PROGRAM MAIN
VAR
	power1,power2,power3,power4: MC_Power;
	axis1,axis2,axis3,axis4: AXIS_REF;
	power1_output,power2_output,power3_output,power4_output:ST_McOutputs;
	

	
	
	move_abs: MC_MoveAbsolute;
	init_pos: LREAL;
	move_init_output:ST_McOutputs;
	
	SetPointGenEnable,SetPointGenEnable1,SetPointGenEnable2,SetPointGenEnable3: MC_ExtSetPointGenEnable;
	SetPointGenDisable,SetPointGenDisable1,SetPointGenDisable2,SetPointGenDisable3: MC_ExtSetPointGenDisable;
	SetPointGenEnable_output,SetPointGenDisable_output,SetPointGenEnable_output1,SetPointGenDisable_output1,SetPointGenEnable_output2,SetPointGenDisable_output2,SetPointGenEnable_output3,SetPointGenDisable_output3:ST_McOutputs;	
	enable,disable:BOOL;
	
	reset_output:ST_McOutputs;
	axis_Reset: MC_Reset;
	
	gen_state:state;
	
	position: LREAL;
	velocity: LREAL;
	direction: DINT;	
	acceleration: LREAL;
	t:LREAL:=0;

	n:UINT:=0;
	a:LINT;
	
	pos1,pos2,pos3,pos4:LREAL;
	acc1,acc2,acc3,acc4:LREAL;
	velo1,velo2,velo3,velo4:LREAL;
	dir: DINT:=1;
	inpos:BOOL:=1;
	flag:UINT:=0;

	flag1: INT;
	ADS_Array: ARRAY[0..12] OF UINT;
	ADS_ParaArray: ARRAY[0..11] OF UINT;
	avar:LREAL;
END_VAR

axis1();(*更新轴状态*)
axis2();(*更新轴状态*)
axis3();(*更新轴状态*)
axis4();(*更新轴状态*)
axis1.ReadStatus();
axis2.ReadStatus();
axis3.ReadStatus();
axis4.ReadStatus();
power();
setpositionGen();
reset();

//move_init();
//TCP/IP receive data
IF NOT GVL.rec_busy THEN
	GVL.bReceive:=TRUE;
END_IF
TCPServer();
IF GVL.number_recdata<>0 THEN
	gen_state:=gen_enable;
	GVL.number_recdata:=0;
	IF GVL.Data_receive[1]>16#7F THEN 
	   GVL.Data_receive[1]:=GVL.Data_receive[1] AND 16#7F;
 	   flag:=1;	
	END_IF
	pos1:=GVL.Data_receive[1];
	pos1:=pos1*256;
	pos1:=(pos1+GVL.Data_receive[2])/10;
	IF flag=1 THEN
		pos1:=-pos1;
		flag:=0;
	END_IF
	velo1:=GVL.Data_receive[3];
	velo1:=velo1*256;
	velo1:=(velo1+GVL.Data_receive[4])/10;
	acc1:=GVL.Data_receive[5];
	acc1:=acc1*256;
	acc1:=(acc1+GVL.Data_receive[6])/10;
	
	IF GVL.Data_receive[7]>16#7F THEN 
	   GVL.Data_receive[7]:=GVL.Data_receive[7] AND 16#7F;
 	   flag:=1;	
	END_IF
	pos2:=GVL.Data_receive[7];
	pos2:=pos2*256;
	pos2:=(pos2+GVL.Data_receive[8])/10;
	IF flag=1 THEN
		pos2:=-pos2;
		flag:=0;
	END_IF
	velo2:=GVL.Data_receive[9];
	velo2:=velo2*256;
	velo2:=(velo2+GVL.Data_receive[10])/10;
	acc2:=GVL.Data_receive[11];
	acc2:=acc2*256;
	acc2:=(acc2+GVL.Data_receive[12])/10;
	
	IF GVL.Data_receive[13]>16#7F THEN 
	   GVL.Data_receive[13]:=GVL.Data_receive[13] AND 16#7F;
 	   flag:=1;	
	END_IF
	pos3:=GVL.Data_receive[13];
	pos3:=pos3*256;
	pos3:=(pos3+GVL.Data_receive[14])/10;
	IF flag=1 THEN
		pos3:=-pos3;
		flag:=0;
	END_IF
	velo3:=GVL.Data_receive[15];
	velo3:=velo3*256;
	velo3:=(velo3+GVL.Data_receive[16])/10;
	acc3:=GVL.Data_receive[17];
	acc3:=acc3*256;
	acc3:=(acc3+GVL.Data_receive[18])/10;
	
	IF GVL.Data_receive[19]>16#7F THEN 
	   GVL.Data_receive[19]:=GVL.Data_receive[19] AND 16#7F;
 	   flag:=1;	
	END_IF
	pos4:=GVL.Data_receive[19];
	pos4:=pos4*256;
	pos4:=(pos4+GVL.Data_receive[20])/10;
	IF flag=1 THEN
		pos4:=-pos4;
		flag:=0;
	END_IF
	velo4:=GVL.Data_receive[21];
	velo4:=velo4*256;
	velo4:=(velo4+GVL.Data_receive[22])/10;
	acc4:=GVL.Data_receive[23];
	acc4:=acc4*256;
	acc4:=(acc4+GVL.Data_receive[24])/10;
END_IF

//ADS receive data
IF ADS_Array[12]=1 THEN
	ADS_Array[12]:=0;
	gen_state:=gen_enable;
	pos1:=ADS_Array[0];
	pos1:=pos1/10;
	velo1:=ADS_Array[1];
	velo1:=velo1/10;
	acc1:=ADS_Array[2];
	acc1:=acc1/10;
	pos2:=ADS_Array[3];
	pos2:=pos2/10;
	velo2:=ADS_Array[4];
	velo2:=velo2/10;
	acc2:=ADS_Array[5];
	acc2:=acc2/10;
	pos3:=ADS_Array[6];
	pos3:=pos3/10;
	velo3:=ADS_Array[7];
	velo3:=velo3/10;
	acc3:=ADS_Array[8];
	acc3:=acc3/10;
	pos4:=ADS_Array[9];
	pos4:=pos4/10;
	velo4:=ADS_Array[10];
	velo4:=velo4/10;
	acc4:=ADS_Array[11];
	acc4:=acc4/10;
END_IF
//ADS updata
avar:=axis1.NcToPlc.ActPos;  //位置
avar:=avar*10;
ADS_ParaArray[0]:= TO_UINT(avar);
avar:=axis1.NcToPlc.Actvelo;  //速度
avar:=avar*10;
ADS_ParaArray[1]:=TO_UINT(avar);
avar:=axis1.NcToPlc.ActAcc;  //加速度
avar:=avar*10;
ADS_ParaArray[2]:=TO_UINT(avar);

avar:=axis2.NcToPlc.ActPos;  //位置
avar:=avar*10;
ADS_ParaArray[3]:= TO_UINT(avar);
avar:=axis2.NcToPlc.Actvelo;  //速度
avar:=avar*10;
ADS_ParaArray[4]:=TO_UINT(avar);
avar:=axis2.NcToPlc.ActAcc;  //加速度
avar:=avar*10;
ADS_ParaArray[5]:=TO_UINT(avar);

avar:=axis3.NcToPlc.ActPos;  //位置
avar:=avar*10;
ADS_ParaArray[6]:= TO_UINT(avar);
avar:=axis3.NcToPlc.Actvelo;  //速度
avar:=avar*10;
ADS_ParaArray[7]:=TO_UINT(avar);
avar:=axis3.NcToPlc.ActAcc;  //加速度
avar:=avar*10;
ADS_ParaArray[8]:=TO_UINT(avar);

avar:=axis4.NcToPlc.ActPos;  //位置
avar:=avar*10;
ADS_ParaArray[9]:= TO_UINT(avar);
avar:=axis4.NcToPlc.Actvelo;  //速度
avar:=avar*10;
ADS_ParaArray[10]:=TO_UINT(avar);
avar:=axis4.NcToPlc.ActAcc;  //加速度
avar:=avar*10;
ADS_ParaArray[11]:=TO_UINT(avar);

CASE gen_state OF
	init:
		power1.Enable:=FALSE;
		power2.Enable:=FALSE;
		power3.Enable:=FALSE;
		power4.Enable:=FALSE;
		SetPointGenEnable.Execute:=FALSE;
		SetPointGenDisable.Execute:=FALSE;
		SetPointGenEnable1.Execute:=FALSE;
		SetPointGenDisable1.Execute:=FALSE;
		SetPointGenEnable2.Execute:=FALSE;
		SetPointGenDisable2.Execute:=FALSE;
		SetPointGenEnable3.Execute:=FALSE;
		SetPointGenDisable3.Execute:=FALSE;
		axis_Reset.Execute:=FALSE;
		gen_state:=gen_power;
			
	gen_power:
		power1.Enable:=TRUE;
		power2.Enable:=TRUE;
		power3.Enable:=TRUE;
		power4.Enable:=TRUE;
		IF power1_output.Done AND power2_output.Done AND power3_output.Done AND power4_output.Done THEN
			gen_state:=gen_move;
		END_IF
		IF axis1.Status.Error OR axis2.Status.Error OR axis3.Status.Error OR axis4.Status.Error THEN
			gen_state := gen_error;
		END_IF
		
	gen_move:
		//	gen_state:=gen_enable;
	gen_enable:

		setpointgenenable.Execute:=TRUE;
		setpointgenenable1.Execute:=TRUE;
		setpointgenenable2.Execute:=TRUE;
		setpointgenenable3.Execute:=TRUE;
		IF SetPointGenEnable.Enabled AND SetPointGenEnable1.Enabled AND SetPointGenEnable2.Enabled AND SetPointGenEnable3.Enabled AND inpos THEN
			flag:=1;
		END_IF

		IF flag=1 THEN
			gen_state:=gen_move;
			IF velo1>1 THEN
				MC_ExtSetPointGenFeed(
					Position:= pos1,		
					Velocity:= velo1, 
					Acceleration:=acc1, 
					Direction:= dir,
					Axis:= axis1);	
			END_IF
			IF velo2>1 THEN
				MC_ExtSetPointGenFeed(
					Position:= pos2,		
					Velocity:= velo2, 
					Acceleration:=acc2, 
					Direction:= dir,
					Axis:= axis2);	
			END_IF
			IF velo3>1 THEN
				MC_ExtSetPointGenFeed(
					Position:= pos3,		
					Velocity:= velo3, 
					Acceleration:=acc3, 
					Direction:= dir,
					Axis:= axis3);
			END_IF	
			IF velo4>1 THEN
				MC_ExtSetPointGenFeed(
					Position:= pos4,		
					Velocity:= velo4, 
					Acceleration:=acc4, 
					Direction:= dir,
					Axis:= axis4);
			END_IF	
		END_IF
		
	//	IF axis1.Status.InTargetPosition AND axis2.Status.InTargetPosition AND axis3.Status.InTargetPosition AND axis4.Status.InTargetPosition AND flag=0 THEN
	//		inpos:=TRUE;
	//	END_IF
		
		IF flag=1 THEN
			flag:=0;
		END_IF

		IF axis1.Status.Error THEN
			gen_state := gen_error;
		END_IF
	
	gen_error:
		SetPointGenEnable.Execute:=FALSE;
		SetPointGenDisable.Execute := SetPointGenEnable.Enabled;	
		SetPointGenEnable1.Execute:=FALSE;
		SetPointGenDisable1.Execute := SetPointGenEnable1.Enabled;
		IF NOT axis1.Status.Coupled THEN
			IF axis1.Status.Error THEN
				gen_state := gen_reset;	
			ELSE
				gen_state := init;
			END_IF
		END_IF
	
	gen_reset:
		axis_Reset.Execute := TRUE;
		SetPointGenDisable.Execute:=FALSE;
		SetPointGenDisable1.Execute:=FALSE;
			
			IF axis_Reset.Done  THEN
				gen_state := init;
			ELSIF axis_Reset.Error  THEN
				gen_state := init; 
			END_IF
		
END_CASE

ACTION move_init:
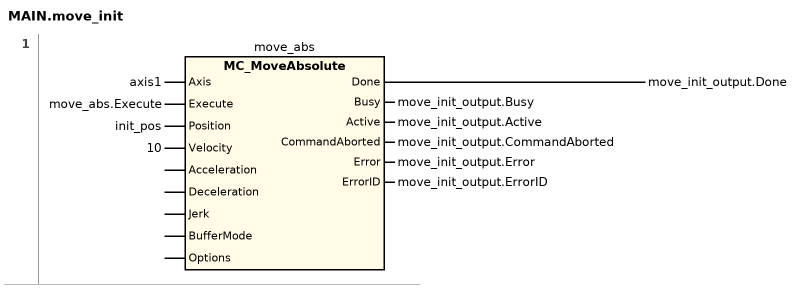
// NETWORK 1
move_abs(
    Axis := axis1,
    Execute := move_abs.Execute,
    Position := init_pos,
    Velocity := 10,
    Busy => move_init_output.Busy,
    Active => move_init_output.Active,
    CommandAborted => move_init_output.CommandAborted,
    Error => move_init_output.Error,
    ErrorID => move_init_output.ErrorID); // MC_MoveAbsolute
move_init_output.Done := move_abs.Done;
END_ACTION

ACTION power:
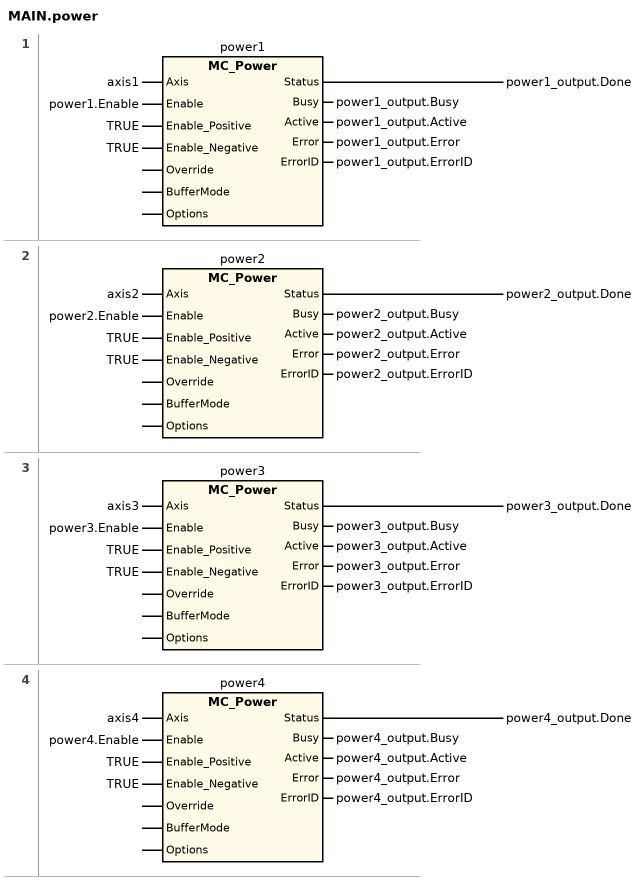
// NETWORK 1
power1(
    Axis := axis1,
    Enable := power1.Enable,
    Enable_Positive := TRUE,
    Enable_Negative := TRUE,
    Busy => power1_output.Busy,
    Active => power1_output.Active,
    Error => power1_output.Error,
    ErrorID => power1_output.ErrorID); // MC_Power
power1_output.Done := power1.Status;

// NETWORK 2
power2(
    Axis := axis2,
    Enable := power2.Enable,
    Enable_Positive := TRUE,
    Enable_Negative := TRUE,
    Busy => power2_output.Busy,
    Active => power2_output.Active,
    Error => power2_output.Error,
    ErrorID => power2_output.ErrorID); // MC_Power
power2_output.Done := power2.Status;

// NETWORK 3
power3(
    Axis := axis3,
    Enable := power3.Enable,
    Enable_Positive := TRUE,
    Enable_Negative := TRUE,
    Busy => power3_output.Busy,
    Active => power3_output.Active,
    Error => power3_output.Error,
    ErrorID => power3_output.ErrorID); // MC_Power
power3_output.Done := power3.Status;

// NETWORK 4
power4(
    Axis := axis4,
    Enable := power4.Enable,
    Enable_Positive := TRUE,
    Enable_Negative := TRUE,
    Busy => power4_output.Busy,
    Active => power4_output.Active,
    Error => power4_output.Error,
    ErrorID => power4_output.ErrorID); // MC_Power
power4_output.Done := power4.Status;
END_ACTION

ACTION reset:
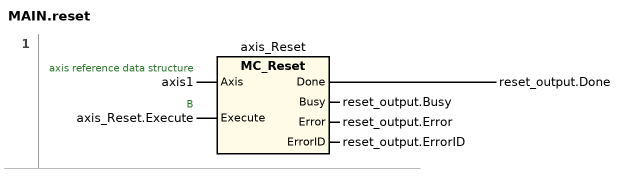
// NETWORK 1
//   axis1: axis reference data structure
//   axis_Reset.Execute: B
axis_Reset(
    Axis := axis1,
    Execute := axis_Reset.Execute,
    Busy => reset_output.Busy,
    Error => reset_output.Error,
    ErrorID => reset_output.ErrorID); // MC_Reset
reset_output.Done := axis_Reset.Done;
END_ACTION

ACTION setpositionGen:
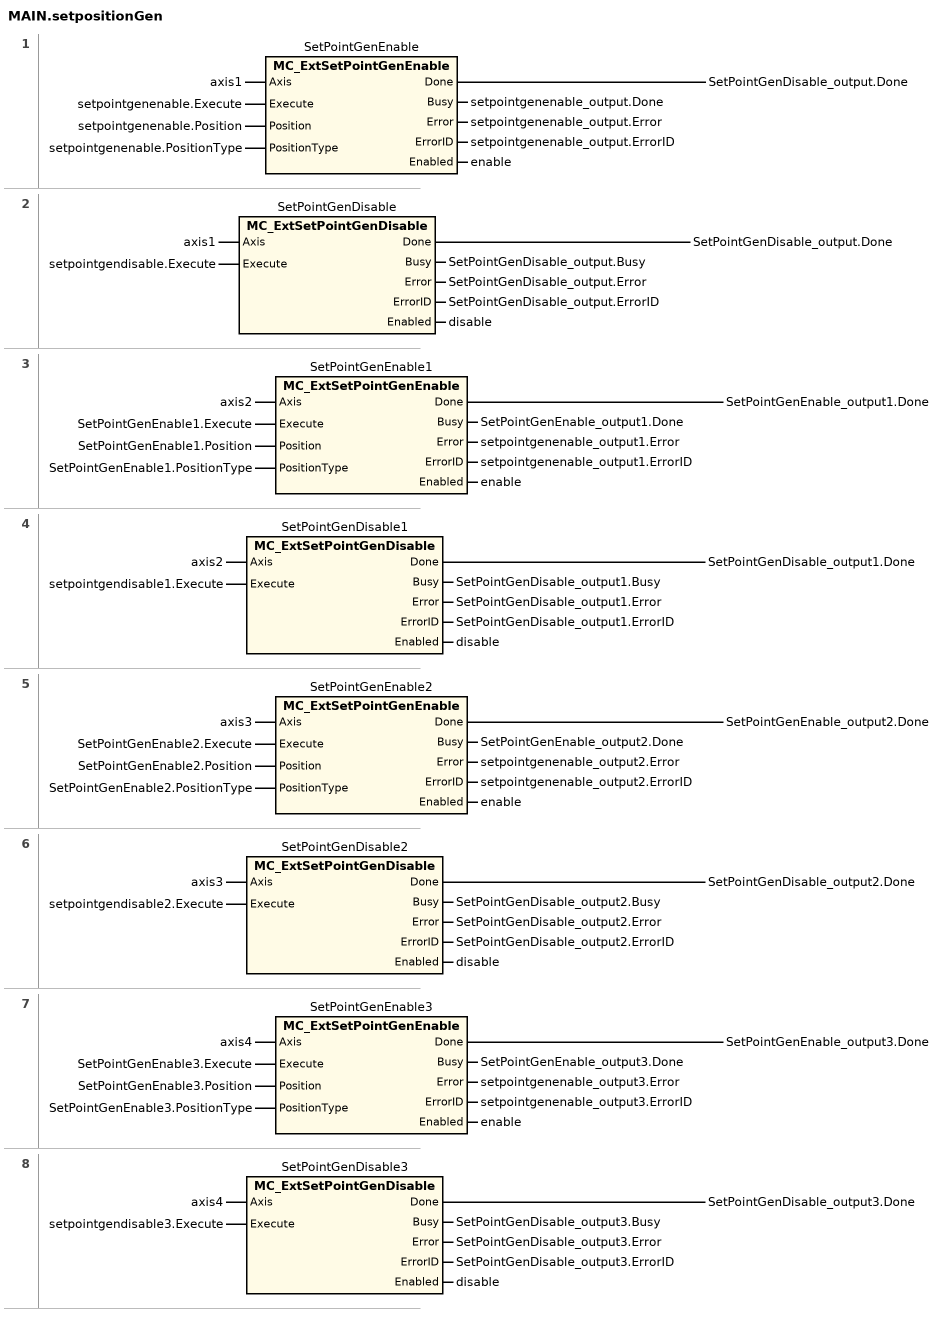
// NETWORK 1
SetPointGenEnable(
    Axis := axis1,
    Execute := setpointgenenable.Execute,
    Position := setpointgenenable.Position,
    PositionType := setpointgenenable.PositionType,
    Busy => setpointgenenable_output.Done,
    Error => setpointgenenable_output.Error,
    ErrorID => setpointgenenable_output.ErrorID,
    Enabled => enable); // MC_ExtSetPointGenEnable
SetPointGenDisable_output.Done := SetPointGenEnable.Done;

// NETWORK 2
SetPointGenDisable(
    Axis := axis1,
    Execute := setpointgendisable.Execute,
    Busy => SetPointGenDisable_output.Busy,
    Error => SetPointGenDisable_output.Error,
    ErrorID => SetPointGenDisable_output.ErrorID,
    Enabled => disable); // MC_ExtSetPointGenDisable
SetPointGenDisable_output.Done := SetPointGenDisable.Done;

// NETWORK 3
SetPointGenEnable1(
    Axis := axis2,
    Execute := SetPointGenEnable1.Execute,
    Position := SetPointGenEnable1.Position,
    PositionType := SetPointGenEnable1.PositionType,
    Busy => SetPointGenEnable_output1.Done,
    Error => setpointgenenable_output1.Error,
    ErrorID => setpointgenenable_output1.ErrorID,
    Enabled => enable); // MC_ExtSetPointGenEnable
SetPointGenEnable_output1.Done := SetPointGenEnable1.Done;

// NETWORK 4
SetPointGenDisable1(
    Axis := axis2,
    Execute := setpointgendisable1.Execute,
    Busy => SetPointGenDisable_output1.Busy,
    Error => SetPointGenDisable_output1.Error,
    ErrorID => SetPointGenDisable_output1.ErrorID,
    Enabled => disable); // MC_ExtSetPointGenDisable
SetPointGenDisable_output1.Done := SetPointGenDisable1.Done;

// NETWORK 5
SetPointGenEnable2(
    Axis := axis3,
    Execute := SetPointGenEnable2.Execute,
    Position := SetPointGenEnable2.Position,
    PositionType := SetPointGenEnable2.PositionType,
    Busy => SetPointGenEnable_output2.Done,
    Error => setpointgenenable_output2.Error,
    ErrorID => setpointgenenable_output2.ErrorID,
    Enabled => enable); // MC_ExtSetPointGenEnable
SetPointGenEnable_output2.Done := SetPointGenEnable2.Done;

// NETWORK 6
SetPointGenDisable2(
    Axis := axis3,
    Execute := setpointgendisable2.Execute,
    Busy => SetPointGenDisable_output2.Busy,
    Error => SetPointGenDisable_output2.Error,
    ErrorID => SetPointGenDisable_output2.ErrorID,
    Enabled => disable); // MC_ExtSetPointGenDisable
SetPointGenDisable_output2.Done := SetPointGenDisable2.Done;

// NETWORK 7
SetPointGenEnable3(
    Axis := axis4,
    Execute := SetPointGenEnable3.Execute,
    Position := SetPointGenEnable3.Position,
    PositionType := SetPointGenEnable3.PositionType,
    Busy => SetPointGenEnable_output3.Done,
    Error => setpointgenenable_output3.Error,
    ErrorID => setpointgenenable_output3.ErrorID,
    Enabled => enable); // MC_ExtSetPointGenEnable
SetPointGenEnable_output3.Done := SetPointGenEnable3.Done;

// NETWORK 8
SetPointGenDisable3(
    Axis := axis4,
    Execute := setpointgendisable3.Execute,
    Busy => SetPointGenDisable_output3.Busy,
    Error => SetPointGenDisable_output3.Error,
    ErrorID => SetPointGenDisable_output3.ErrorID,
    Enabled => disable); // MC_ExtSetPointGenDisable
SetPointGenDisable_output3.Done := SetPointGenDisable3.Done;
END_ACTION

END_PROGRAM

(* stored: Version 1.1.0.1, ProductVersion 3.1.4024.15
   POU MAIN: Id {b5f9f374-b168-4801-9ce4-b8c4d83c90ee}, SpecialFunc None
   Action move_init: Id {06a47df9-86bb-4d08-9c86-083a0f773e80}
   Action power: Id {8b469144-5c09-487e-8637-7d166d37593e}
   Action reset: Id {d4c531c5-ab2c-485e-947c-8ec7bbf86e8a}
   Action setpositionGen: Id {92c8d64b-13a0-40cc-90b1-01eed4cbedc3} *)
